FUNCTION CONVERT_MASS_TO_FLOW : REAL
VAR_INPUT
	Mass:REAL; (*in gramme*)
	Delay:TIME; (*in ms*)
END_VAR
VAR
END_VAR

CONVERT_MASS_TO_FLOW:=Mass/TIME_TO_DWORD(Delay)*60000;

END_FUNCTION

(* stored: Version 1.1.0.1, ProductVersion 3.1.0.26
   POU CONVERT_MASS_TO_FLOW: Id {e0406e27-9b33-49ff-a751-f6255274c4b9} *)
